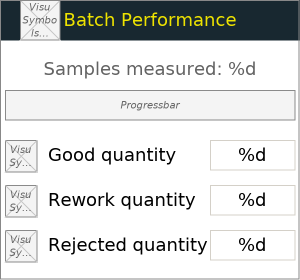
VISUALIZATION AOIBatchPerformanceFrame  // 300x280
VAR_IN_OUT
	stBatchPerformanceFrame : ST_BatchPerformacne;
END_VAR
    Label (45,140 160x30), "Good quantity"
    Label (45,185 160x30), "Rework quantity"
    Label (45,230 160x30), "Rejected quantity"
    Image (5,230 32x32), image: VisuSymbols.Symbols.Wrong
    Image (5,140 32x32), image: VisuSymbols.Symbols.OK
    Image (5,185 32x32), image: VisuSymbols.Symbols.ArrowRoundLeftUp
    Textfield (210,140 85x30), "%d", text variable: stBatchPerformanceFrame.iGoodQuantity
    Textfield (210,185 85x30), "%d", text variable: stBatchPerformanceFrame.iReworkQuantity
    Textfield (210,230 85x30), "%d", text variable: stBatchPerformanceFrame.iRejectedQuantity
    Rectangle (0,0 300x40), "Batch Performance"
    Progressbar (5,90 290x30), variable: stBatchPerformanceFrame.iBatchProgress
    Rectangle (25,54 250x30), "Samples measured: %d", text variable: stBatchPerformanceFrame.iCurrentQuantity
    Image (20,0 40x40), image: VisuSymbols.Symbols.MonitorCurve
END_VISUALIZATION

(* stored: Version 1.1.0.1, ProductVersion 3.1.4024.9
   Visu AOIBatchPerformanceFrame: Id {f63fd335-348b-4f40-b691-a7df547d6194} *)
